FUNCTION AddCounterToMessage : T_MaxString
VAR_INPUT
	counter : INT;
	message : T_MaxString;
END_VAR
VAR
END_VAR

AddCounterToMessage := CONCAT('CRISTART ', 
					   CONCAT(INT_TO_STRING(counter), 
					   CONCAT(' ',
					   CONCAT(message, 
							 ' CRIEND'))));

END_FUNCTION

(* stored: Version 1.1.0.1, ProductVersion 3.1.4024.12
   POU AddCounterToMessage: Id {f098f86f-3ce0-4325-936e-91ba26331161}, SpecialFunc None *)
